// TIA Portal V19 export
DATA_BLOCK "A0301_Manager"   // DB23
// stored: InstanceOfName A0301_Manager_FB, InstanceOfType FB
"A0301_Manager_FB"
   // VAR_INPUT
   //    AreaInterface : "AreaInterface";
   //    DataIn : Struct
   //       SemiAut_Pb : Bool;
   //       P1 : Struct
   //          Sens_Ing : Array[1..3] of Bool;
   //          Sens_Out : Array[1..3] of Bool;
   //       END_STRUCT;
   //       P2 : Struct
   //          Sens_Ing : Array[1..3] of Bool;
   //          Sens_Out : Array[1..3] of Bool;
   //       END_STRUCT;
   //       P3 : Struct
   //          Sens_Ing : Array[1..3] of Bool;
   //          Sens_Out : Array[1..3] of Bool;
   //       END_STRUCT;
   //       P4 : Struct
   //          Sens_Ing : Array[1..3] of Bool;
   //          Sens_Out : Array[1..3] of Bool;
   //       END_STRUCT;
   //       P5 : Struct
   //          Sens_Fuori_Ingombro_A0301 : Bool;
   //       END_STRUCT;
   //    END_STRUCT;
   //    CIn : Struct
   //       Trasporto : "SpeedMachine_COut";
   //       P1 : Struct
   //          Fermi : "ValveMachine_COut";
   //          Sfalsatore : "ValveMachine_COut";
   //       END_STRUCT;
   //       P2 : Struct
   //          Fermi : "ValveMachine_COut";
   //          Sollevatore : "ValveMachine_COut";
   //       END_STRUCT;
   //       P3 : Struct
   //          Fermi : "ValveMachine_COut";
   //       END_STRUCT;
   //       P4 : Struct
   //          Fermi : "ValveMachine_COut";
   //       END_STRUCT;
   //       P5 : Struct
   //          Sollevatori { ExternalAccessible := 'False'; ExternalVisible := 'False'; ExternalWritable := 'False'} : "ValveMachine_COut";
   //          Spintore_Lat : Struct
   //             Spin_Lat1 : Struct
   //                Standstill : Bool;
   //                Rest_CheckNext : Bool;
   //                Work_CheckNext : Bool;
   //                Rest : Bool;
   //                Work : Bool;
   //             END_STRUCT;
   //             Spin_Lat2 : Struct
   //                Standstill : Bool;
   //                Rest_CheckNext : Bool;
   //                Work_CheckNext : Bool;
   //                Rest : Bool;
   //                Work : Bool;
   //             END_STRUCT;
   //             Vrt_1 : "ValveMachine_COut";
   //             Orz_1 : "ValveMachine_COut";
   //             Vrt_2 : "ValveMachine_COut";
   //             Orz_2 : "ValveMachine_COut";
   //          END_STRUCT;
   //          SpintoreLong { ExternalAccessible := 'False'; ExternalVisible := 'False'; ExternalWritable := 'False'} : Struct
   //             Ax : "Positioning_EPOS_Machine_COut";
   //             Vert : "ValveMachine_COut";
   //          END_STRUCT;
   //          SensUscitaBanco : Bool;
   //       END_STRUCT;
   //       Ribaltatore : Struct
   //          Solleva_Rib : "ValveMachine_COut";
   //          Ax : "Positioning_EPOS_Machine_COut";
   //          Sts_Ribaltatore : Struct
   //             Pos0_Reached : Bool;
   //             Pos1_Reached : Bool;
   //             Pos2_Reached : Bool;
   //             Pos3_Reached : Bool;
   //          END_STRUCT;
   //       END_STRUCT;
   //       SpintoreLong : Struct
   //          Ax_Sts { ExternalAccessible := 'False'; ExternalVisible := 'False'; ExternalWritable := 'False'} : Struct
   //             PosAttesa_Reached : Bool;
   //             PosFineSpinta_Reached : Bool;
   //          END_STRUCT;
   //          Spin_Ev : "ValveMachine_COut";
   //       END_STRUCT;
   //       ProdManager : "Prod_Beam_Ctrl";
   //    END_STRUCT;
   // END_VAR
   // VAR_OUTPUT
   //    MachineInterface : "MachineInterface";
   //    COut : Struct
   //       P1 : Struct
   //          Fermi : "ValveMachine_Manager";
   //          Pareggiatore : "ValveMachine_Manager";
   //          ReqPTrk_A02 : Bool;
   //       END_STRUCT;
   //       P2 : Struct
   //          Fermi : "ValveMachine_Manager";
   //          Sollevatore : "ValveMachine_Manager";
   //       END_STRUCT;
   //       P3 : Struct
   //          Fermi : "ValveMachine_Manager";
   //       END_STRUCT;
   //       P4 : Struct
   //          Fermi : "ValveMachine_Manager";
   //       END_STRUCT;
   //       P5 : Struct
   //          Spintore_Lat_1 { ExternalAccessible := 'False'; ExternalVisible := 'False'; ExternalWritable := 'False'} : "ValveMachine_Manager";
   //          Spintore_Lat_2 { ExternalAccessible := 'False'; ExternalVisible := 'False'; ExternalWritable := 'False'} : "ValveMachine_Manager";
   //          Sollevatori : "ValveMachine_Manager";
   //       END_STRUCT;
   //       Trasporto : "SpeedMachine_CIn_Manager";
   //       Trasporto_Brw_Req : Bool;
   //       Trasporto_Frw_Req : Bool;
   //       Ribaltatore : Struct
   //          Solleva : "ValveMachine_Manager";
   //          Ax : "Positioning_EPOS_Machine_Manager";
   //          Ax_Req : Struct
   //             Pos0 : Bool;
   //             Pos1 : Bool;
   //             Pos2 : Bool;
   //             Pos3 : Bool;
   //          END_STRUCT;
   //          Solleva_REST_Req : Bool;
   //          Solleva_WORK_Req : Bool;
   //       END_STRUCT;
   //    END_STRUCT;
   // END_VAR
   // VAR_IN_OUT
   //    Par : Struct
   //       DlySensorsON : Time;
   //       DlySensorsOFF : Time;
   //       TRK : Struct
   //          BTrk_MoveP4Exit : Time;
   //          BTrk_MoveToP5 : Time;
   //       END_STRUCT;
   //    END_STRUCT;
   //    Data : Struct
   //       LastCounter_PartMove_P2toP4 : LReal;
   //       LastCounter_PartMove_P1toP2 : LReal;
   //       LastCounter_PartMove_P1toP3 : LReal;
   //    END_STRUCT;
   // END_VAR
   // VAR
   //    Alarm : Struct
   //       WrongShiftDone { S7_SetPoint := 'True'} : Bool;
   //       P2toP4_NotReached : Bool;
   //       P1toP2_NotReached : Bool;
   //       P1toP3_NotReached : Bool;
   //       PTrk_TO_BTrk : Struct
   //          Status : USInt;
   //       END_STRUCT;
   //       STOP_FineTurno : Bool;
   //       STOP_End_Of_Proroduction : Bool;
   //       STOP_ControlloQualita : Bool;
   //    END_STRUCT;
   //    Sts : Struct
   //       SemiAut : Struct
   //          ON : Bool;
   //          Request : Bool;
   //          MaterialFrw : Bool;
   //       END_STRUCT;
   //       P1 : Struct
   //          Fermi : Struct
   //             Sens_Ing : Bool;
   //             Sens_Out : Bool;
   //          END_STRUCT;
   //          Sfalsatura_OK : Bool;
   //       END_STRUCT;
   //       P2 : Struct
   //          Fermi : Struct
   //             Some_Sens_Ing : Bool;
   //             Sens_Ing : Bool;
   //             Sens_Out : Bool;
   //          END_STRUCT;
   //       END_STRUCT;
   //       P3 : Struct
   //          Fermi : Struct
   //             Some_Sens_Ing : Bool;
   //             Sens_Ing : Bool;
   //             Sens_Out : Bool;
   //          END_STRUCT;
   //       END_STRUCT;
   //       P4 : Struct
   //          Fermi : Struct
   //             Some_Sens_Ing : Bool;
   //             Sens_Ing : Bool;
   //             Sens_Out : Bool;
   //          END_STRUCT;
   //       END_STRUCT;
   //       A0301_Station1 : Struct
   //          ZoneEmpty { ExternalAccessible := 'False'; ExternalVisible := 'False'; ExternalWritable := 'False'} : Bool;
   //          Trk { ExternalAccessible := 'False'; ExternalVisible := 'False'; ExternalWritable := 'False'} : Struct
   //             Actual_O_ID : DInt;
   //             OLD_OID : DInt;
   //             A0301_PTrk_Absence : Bool;
   //             A0301_BTrk_Absence : Bool;
   //             Wait_A0301_Recive : Bool;
   //          END_STRUCT;
   //       END_STRUCT;
   //       Attrezzamento : Struct
   //          Ready : Bool;
   //          FindNewID : Bool;
   //          RequestNewPosition : Bool;
   //          OLD_OID : DInt;
   //       END_STRUCT;
   //       AlarmsPresence : Bool;
   //       WarningsPresence : Bool;
   //       IsStandstill : Bool;
   //    END_STRUCT;
   //    Ctrl : Struct
   //       Stop : Bool;
   //       TRK : Struct
   //          PTrk : Struct
   //             Start_Brw : Bool;
   //             Start_Frw : Bool;
   //             Pos1_TO_Pos3 : Bool;
   //             Pos1_TO_Pos2 : Bool;
   //             Pos2Entry_TO_Pos2Solleva : Bool;
   //             Paregg_Pos1_to_Pos2 : Bool;
   //             Paregg_Pos1_to_Pos3 : Bool;
   //          END_STRUCT;
   //          BTrk : Struct
   //             Pos2Up_TO_Pos2Down : Bool;
   //             WritePos2Up_TO_Pos2Down : Bool;
   //             Pos4_Entry_TO_Pos4_Exit : Bool;
   //             Pos4_Entry_Cndz_To_Exit : Bool;
   //             Pos4_Exit_TO_Pos4_to_Pos5 : Bool;
   //             Pos4_to_Pos5_TO_Pos5_Lat_Spin_Orz : Struct
   //                Exe : Bool;
   //                Solleva : Bool;
   //                Trasla : Bool;
   //             END_STRUCT;
   //             Pos5_SpinLat_TO_Pos5_SpinLong : Bool;
   //          END_STRUCT;
   //          Ribaltatore : Struct
   //             MoveToPos0 : Bool;
   //             MoveToPos1 : Bool;
   //             MoveToPos2 : Bool;
   //             MoveToPos3 : Bool;
   //          END_STRUCT;
   //       END_STRUCT;
   //       P1 : Struct
   //          Fermi : Struct
   //             Rest : Bool;
   //             Work : Bool;
   //          END_STRUCT;
   //          Pareggiatore : Struct
   //             Rest : Bool;
   //             Work : Bool;
   //          END_STRUCT;
   //          PartMove_P1toP3_Init : Bool;
   //          PartMove_P1toP2_Init : Bool;
   //       END_STRUCT;
   //       P2 : Struct
   //          Fermi : Struct
   //             Rest : Bool;
   //             Work : Bool;
   //          END_STRUCT;
   //          Sollevatore : Struct
   //             EnableMove : Bool;
   //             Rest : Bool;
   //             Work : Bool;
   //          END_STRUCT;
   //          PartMove_P2toP4_Init : Bool;
   //       END_STRUCT;
   //       P3 : Struct
   //          Fermi : Struct
   //             Rest : Bool;
   //             Work : Bool;
   //          END_STRUCT;
   //       END_STRUCT;
   //       P4 : Struct
   //          Fermi : Struct
   //             Rest : Bool;
   //             Work : Bool;
   //          END_STRUCT;
   //          Part_Move_P2toP4_Init : Bool;
   //       END_STRUCT;
   //       P5 : Struct
   //          Spintore_Lat_1 : Struct
   //             Rest : Bool;
   //             Work : Bool;
   //          END_STRUCT;
   //          Spintore_Lat_2 : Struct
   //             Rest : Bool;
   //             Work : Bool;
   //          END_STRUCT;
   //          Sollevatori : Struct
   //             Rest : Bool;
   //             Work : Bool;
   //          END_STRUCT;
   //       END_STRUCT;
   //       Ribaltatore : Struct
   //          Solleva : Struct
   //             EnableMove : Bool;
   //             Rest : Bool;
   //             Work : Bool;
   //          END_STRUCT;
   //       END_STRUCT;
   //    END_STRUCT;
   //    Ctrl_Part_Move_P1toP2 : "Check_Part_Movement";
   //    Ctrl_Part_Move_P1toP3 { S7_SetPoint := 'True'} : "Check_Part_Movement";
   //    Ctrl_Part_Move_P2toP4 : "Check_Part_Movement";
   //    TON_Stop { S7_SetPoint := 'True'} : IEC_TIMER;
   //    TON : Struct
   //       BTrk_MoveP4Exit : TON_TIME;
   //       BTrk_MoveToP5 : TON_TIME;
   //       Delay_Pos1Ribalta { S7_SetPoint := 'True'} : TON_TIME;
   //       P1 : Struct
   //          Sens_Ing : Struct
   //             DelayOn : TON_TIME;
   //          END_STRUCT;
   //          Sens_Out : Struct
   //             DelayOff : TOF_TIME;
   //          END_STRUCT;
   //       END_STRUCT;
   //       P2 : Struct
   //          Sens_Ing : Struct
   //             DelayOn : TON_TIME;
   //          END_STRUCT;
   //          Sens_Out : Struct
   //             DelayOff : TOF_TIME;
   //          END_STRUCT;
   //       END_STRUCT;
   //       P3 : Struct
   //          Sens_Ing : Struct
   //             DelayOn : TON_TIME;
   //          END_STRUCT;
   //          Sens_Out : Struct
   //             DelayOff : TOF_TIME;
   //          END_STRUCT;
   //       END_STRUCT;
   //       P4 : Struct
   //          Sens_Ing : Struct
   //             DelayOn : TON_TIME;
   //          END_STRUCT;
   //          Sens_Out : Struct
   //             DelayOff : TOF_TIME;
   //          END_STRUCT;
   //       END_STRUCT;
   //       P1_Exit_P3 : IEC_TIMER;
   //       P1_Exit_P2 : IEC_TIMER;
   //    END_STRUCT;
   //    HMI : Struct
   //       B_ResetShiftDone : Bool;
   //    END_STRUCT;
   //    AUX : Struct
   //       SemiAut_Pb : Bool;
   //       B_ResetShiftDone : Bool;
   //    END_STRUCT;
   //    BTrk_Item : Struct
   //       O_ID : DInt;
   //       BLean : Real;
   //       W_A : Real;
   //       H_B : Real;
   //       Tol_Max : Real;
   //       Tol_Min : Real;
   //       Good { ExternalAccessible := 'False'; ExternalVisible := 'False'; ExternalWritable := 'False'} : Bool;
   //       Bad { ExternalAccessible := 'False'; ExternalVisible := 'False'; ExternalWritable := 'False'} : Bool;
   //    END_STRUCT;
   //    PLen_Pos1 : Real;
   //    PLen_Pos3 : Real;
   // END_VAR
BEGIN
END_DATA_BLOCK
